FUNCTION_BLOCK SORT_CTL (* Peg/Ring Sort Control *)
  (* Standard: 61499 ITA; Classification: Testbed *)
  (* Version 0.1, 2004-08-06, JHC, Rockwell Automation, Added RING_LOST. *)
  (* Version 0.0, 2002-05-08, JHC, Rockwell Automation *)
  (* Compiler header: package fb.rt.ita.testbed; *)
  (* Compiler Java Sun JDK 1.4.2 *)
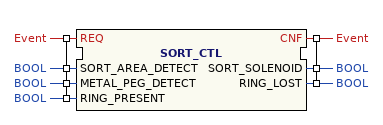
  EVENT_INPUT
    REQ WITH METAL_PEG_DETECT, SORT_AREA_DETECT, RING_PRESENT;
  END_EVENT
  EVENT_OUTPUT
    CNF WITH SORT_SOLENOID, RING_LOST;
  END_EVENT
  VAR_INPUT
    SORT_AREA_DETECT : BOOL;
    METAL_PEG_DETECT : BOOL;
    RING_PRESENT : BOOL;
  END_VAR
  VAR_OUTPUT
    SORT_SOLENOID : BOOL;
    RING_LOST : BOOL; (* Ring passed by sorter without deflection because chute was full *)
  END_VAR
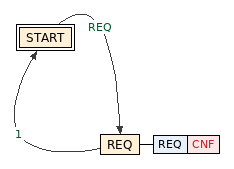
  EC_STATES
    START;
    REQ : REQ -> CNF;
  END_STATES
  EC_TRANSITIONS
    START TO REQ := REQ;
    REQ TO START := 1;
  END_TRANSITIONS
  ALGORITHM REQ IN LD:
    SORT_SOLENOID := METAL_PEG_DETECT ! SORT_AREA_DETECT & RING_PRESENT ! &;
    RING_LOST := METAL_PEG_DETECT ! SORT_AREA_DETECT & RING_PRESENT &;
  END_ALGORITHM
END_FUNCTION_BLOCK
